FUNCTION_BLOCK FB_MotorsReset
VAR_INPUT
	bExecute : BOOL;
END_VAR
VAR_OUTPUT
	bDone : BOOL;
	bError: BOOL;
	bBusy : BOOL;
END_VAR
VAR_IN_OUT
	Axis : AXIS_REF;
END_VAR
VAR
	fbReset	: MC_Reset;
	bReset	: BOOL := TRUE;

END_VAR

//Axis Reset
IF bExecute THEN
	fbReset(Axis := Axis, Execute := bReset, Done => bDone, Error => bError, Busy => bBusy);
END_IF
IF bDone THEN
	bReset := FALSE;
END_IF

METHOD Reset : BOOL
VAR_INPUT
END_VAR
bReset := TRUE;
Reset := bReset;
END_METHOD

END_FUNCTION_BLOCK

(* stored: Version 1.1.0.1, ProductVersion 3.1.4024.12
   POU FB_MotorsReset: Id {7a3e4215-b5be-40fe-b889-7d70a5148238}, SpecialFunc None
   Method Reset: Id {b9304837-371d-411d-8cb8-12a541f16836} *)
